{attribute 'qualified_only'}
VAR_GLOBAL
	Max_50kVChargerVoltage : REAL := 50000; //50kV
	Min_50kVChargerVoltage : REAL := 0;
	
	Max_50kVChargerCurrent : REAL := 0.18; //total peak charge current is 0.18A
	Min_50kVChargerCurrent : REAL := 0;
	
	Max_12kVChargerVoltage : REAL := 12000; //12kV
	Min_12kVChargerVoltage : REAL := 0;
	
	Max_12kVChargerCurrent : REAL := 0.75; //total peak charge current is 0.75A
	Min_12kVChargerCurrent : REAL := 0;
	
	Max_30kVChargerVoltage : REAL := 30000; //30kV
	Min_30kVChargerVoltage : REAL := 0;
	
	Max_30kVChargerCurrent : REAL := 0.6; //total peak charge current is 0.6A
	Min_30kVChargerCurrent : REAL := 0;	
	//Max_GLS1_ChargerV	   : REAL := 50000; //form trigger
	//Max_GLS2_ChargerV	   : REAL := 50000; // preform trigger
	//Max_GLS3_ChargerV	   : REAL := 30000; // preform cap charger
	
	Max_CapVoltage			: REAL := 32000;  //assuming 32kV cap....  
	Min_CapVoltage			: REAL := 0;
	
	UpperLimit12kVCaps		: REAL := 10500; 
	//LowerLimit12kVCaps	: REAL := -2000;
	UpperLimit50kVCaps		: REAL := 35000; 
	
	(*ULimit_PeakCapRequiredV	: REAL := 10000; //10kV veto
	LLimit_PeakCapRequiredV	: REAL := -2000; //-2kV
	ULimit_SustCapRequiredV	: REAL := 12000; //12kv veto
	LLimit_SustCapRequiredV	: REAL := -2000; //-2kv
	ULimit_FormCapRequiredV : REAL := 35000;
	LLimit_FormCapRequiredV : REAL := 0;
	*)
	//ULimit_PreFormCapRequiredV : REAL := 30000; //gls3
	//LLimit_PreFormCapRequiredV : REAL := 0;
		
END_VAR

(* stored: Version 1.1.0.1, ProductVersion 3.1.4024.11
   GVL EngVal: Id {279758fb-6686-4086-920b-c14098f79a19} *)
